TYPE "Changeover_ShW"
VERSION : 0.1
   STRUCT
      AutoDownloadTrigger : Bool;
      ManualDownloadTrigger : Bool;
      Result : Int;
      Completed : Bool;
   END_STRUCT;

END_TYPE

